Universal Robots PolyScope program: test_circ_motion7.urp

Program test_circ_motion7 (installation=default directory=/programs createdIn=5.14.5 lastSavedIn=5.14.5 robotSerialNumber=20236801216)
Calibrated DH parameters: a=[-0.000021, -0.748897, -0.28186, -0.00004, -0.000055, 0]; d=[0.236225, -424.082933, -1564.66872, 1988.95162, 0.159094, 0.153873]; alpha=[1.570844, 0.001002, 0.000337, 1.571488, -1.569996, 0]; deltaTheta=[0, -0.516316, 5.626292, 1.173211, 0.000001, 0]
InitVariablesNode
Robot Program (runOnlyOnce=true)
  Script file /programs/convert_headingxplus_axang.script
    | # this script is a function.
    | # inputs: heading ccw from x+ axis (in radians)
    | # outputs: rxout, ryout, rzout
    | 
    | 
    | 
    | # list of variables used
    | # heading
    | # axisxraw, axisyraw, axiszraw, magnitude, axisxunit, axisyunit, axiszunit, angle
    | # rxout, ryout, rzout
    | 
    | def convert_to_axang(heading):
    |  axisxraw = -1 * sin(heading)
    |  axisyraw = cos(heading) + 1
    |  axiszraw = sin(heading)
    | 
    |  magnitude = sqrt(axisxraw*axisxraw + axisyraw*axisyraw + axiszraw*axiszraw)
    | 
    |  axisxunit = axisxraw / magnitude
    |  axisyunit = axisyraw / magnitude
    |  axiszunit = axiszraw / magnitude
    | 
    |  angle = acos( (cos(heading) - 1) / 2 )
    | 
    |  rxout = axisxunit * angle
    |  ryout = axisyunit * angle
    |  rzout = axiszunit * angle
    | 
    |  return [rxout, ryout, rzout]
    | end
  Script file /programs/test_convertheadingxplus.script
    | # this script is a test motion program to use convert_headingxplus_axang.script and see if that works
    | pi = 3.1415926535
    | 
    | p1 = p[-.80,.9,0,pi/2,0,0]
    | 
    | movej(p1, a=1.2, v=0.25)
    | 
    | heading = 270 * pi/180
    | 
    | # call script
    | ret = convert_to_axang()
    | 
    | p2 = p[p1[0], p1[1], p1[2], ret[0], ret[1], ret[2]]
    | 
    | movej(p2, a=1.2, v=0.25)
    | 
    | # position 2
    | heading = 225 * pi/180
    | ret = convert_to_axang()
    | p2 = p[p1[0], p1[1], p1[2], ret[0], ret[1], ret[2]]
    | movej(p2, a=1.2, v=0.25)
    | 
    | # position 3
    | heading = 180 * pi/180
    | convert_to_axang()
    | ret = p3 = p[p1[0], p1[1], p1[2], ret[0], ret[1], ret[2]]
    | movej(p3, a=1.2, v=0.25)
